FUNCTION_BLOCK SimpleTimeRecorder
VAR_INPUT
END_VAR
VAR_OUTPUT
END_VAR
VAR
  _duration_in_ms: ULINT;
  _timestamp_in_ms: ULINT;
END_VAR

{attribute 'monitoring' := 'call'}
PROPERTY act_duration_in_ms : ULINT
GET
IF timestamp_in_ms > 0 THEN
  act_duration_in_ms := act_timestamp_in_ms - timestamp_in_ms;
ELSE
  act_duration_in_ms := duration_in_ms;
END_IF
END_GET
END_PROPERTY

{attribute 'monitoring' := 'call'}
PROPERTY PRIVATE act_timestamp_in_ms : ULINT
GET
act_timestamp_in_ms := F_GetSystemTime() / 10000;
END_GET
END_PROPERTY

METHOD PRIVATE apply_duration
VAR_INPUT
END_VAR
IF timestamp_in_ms > 0 THEN
  duration_in_ms := act_duration_in_ms;
  timestamp_in_ms := 0;
END_IF
END_METHOD

{attribute 'monitoring' := 'call'}
PROPERTY duration : TIME
GET
duration := TO_TIME(duration_in_ms);
END_GET
END_PROPERTY

{attribute 'monitoring' := 'call'}
PROPERTY PUBLIC duration_in_ms : ULINT
GET
duration_in_ms := _duration_in_ms;
END_GET
SET
_duration_in_ms := duration_in_ms;
END_SET
END_PROPERTY

METHOD record
VAR_INPUT
  execute: BOOL;
END_VAR
VAR_INST
  r_signal: R_TRIG;
  r_execute: R_TRIG;
  f_execute: F_TRIG;
END_VAR
r_execute(CLK:=execute);
f_execute(CLK:=execute);
IF r_execute.Q THEN
  timestamp_in_ms := act_timestamp_in_ms;
END_IF
IF f_execute.Q THEN
  apply_duration();
END_IF
END_METHOD

METHOD reset
VAR_INPUT
END_VAR
duration_in_ms := 0;
timestamp_in_ms := 0;
END_METHOD

{attribute 'monitoring' := 'call'}
PROPERTY PUBLIC timestamp_in_ms : ULINT
GET
timestamp_in_ms := _timestamp_in_ms;
END_GET
SET
_timestamp_in_ms := timestamp_in_ms;
END_SET
END_PROPERTY

END_FUNCTION_BLOCK

(* stored: Version 1.1.0.1, ProductVersion 3.1.4024.9
   POU SimpleTimeRecorder: Id {e5f908a6-1d21-029a-2e15-c522870cbaaa}, SpecialFunc None
   Property act_duration_in_ms: Id {b06090b1-1ca5-04d7-2ec6-a2ce3bd105bc}
   Get Get: Id {b8168a9b-2159-0145-0bd7-78f27443161c}
   Property act_timestamp_in_ms: Id {7ddbc0ef-bf35-0d0f-2415-5110fd05b7e5}
   Get Get: Id {aecfedff-00f5-0b03-0432-6b4d707a7a27}
   Method apply_duration: Id {a33e2165-65fb-0af5-3822-ce3728e366da}
   Property duration: Id {24846e4a-c2d9-0962-234a-24735cb729f2}
   Get Get: Id {88b45260-dc7d-06f6-0150-1e84dbb63d3e}
   Property duration_in_ms: Id {c3e03a26-ec18-0900-1bf3-4dc359a9377b}
   Get Get: Id {9d615a78-6aa7-0ffc-08ad-e3ab7e6bc574}
   Set Set: Id {8d9da77b-6b79-0045-21c6-0ffd76bf87fb}
   Method record: Id {8ef85350-afd8-0be6-11c0-55116fb94f85}
   Method reset: Id {08509da3-ed68-015b-0642-47cbbc9096f7}
   Property timestamp_in_ms: Id {d67fa0b8-d19e-0ba8-24c6-be9675dbf922}
   Get Get: Id {6f2ef54a-d726-0dd3-36fb-fa7f0783bfa9}
   Set Set: Id {a5dd66c9-cb2d-0605-35ef-1646691b3dbe} *)
